PROGRAM MAIN
VAR
END_VAR

END_PROGRAM

(* stored: Version 1.1.0.1
   POU MAIN: Id {51da1b52-2b53-44ea-a693-73c155047262} *)
